PROGRAM Motion
VAR
	Power : MC_Power;
	Speed : MC_Jog;
	Velocity : MC_MoveVelocity;
	
END_VAR

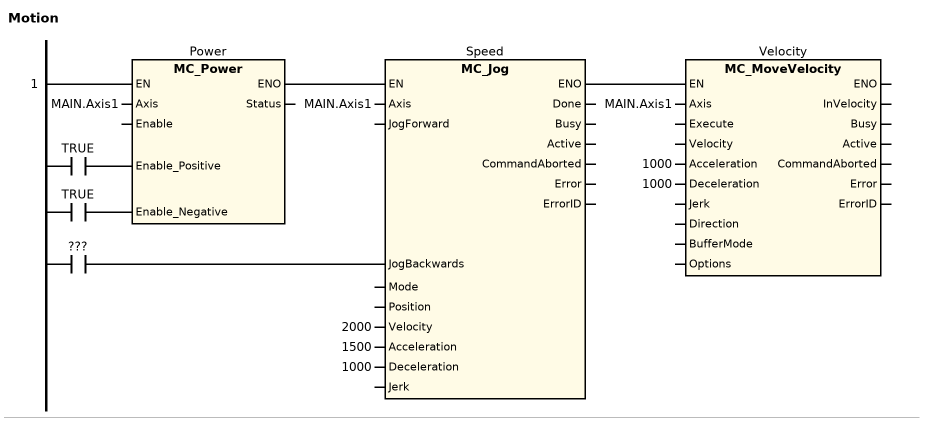
// NETWORK 1
Power(Axis := MAIN.Axis1, Enable_Positive := TRUE, Enable_Negative := TRUE); // MC_Power
Speed(Axis := MAIN.Axis1, Velocity := 2000, Acceleration := 1500, Deceleration := 1000); // MC_Jog
Velocity(Axis := MAIN.Axis1, Acceleration := 1000, Deceleration := 1000); // MC_MoveVelocity

END_PROGRAM

(* stored: Version 1.1.0.1, ProductVersion 3.1.4024.13
   POU Motion: Id {61f7a26d-06ec-4607-a4d7-e9515f747e29}, SpecialFunc None *)
